# B&R Automation Studio project ciclicheskoe11
Automation Studio 4.5.2.102; technology packages: Acp10Arnc0 1.0.0

## Configuration Config1

CPU 4PP065.0571-P74, AutomationRuntime D4.52, Build 4.1.2, Vc V4.52.0

### Task classes (Cpu.sw)
```
Cyclic#1:
  RobotContr <- RobotControl.prg
DataObjects: Acp10sys
Binaries: TCData, vcfile, vcfntttf, vcpfmtcx, arial, vcmgr, vccovl, vcdsint, vcpdpp30, vcshared, vcpfpp30, vcpdsw, vcalarm, vccbtn, vcptelo, vcgclass, vcdsloc, arialbd, vcrt, Visu02, vctcal, Visu01, Visu03, vcbclass, udbdef, vcctext, vccbmp, vcchspot, vccnum, ashwac, arconfig, User, sysconf, iomap, asfw, ashwd, Role, acp10cfg, Acp10map
Libraries: Acp10sdc, URTK_lib, Acp10man, Acp10par, NcGlobal, asstring, powerlnk, astime, fileio, runtime, dataobj, vcresman, Library
```

### Hardware
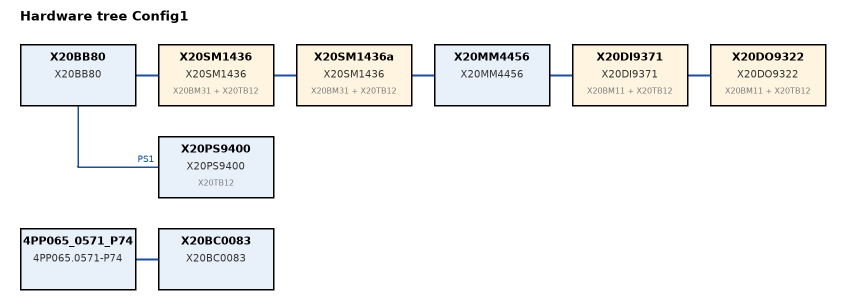
```
4PP065_0571_P74 : 4PP065.0571-P74 v1.1.2.0
  Connector IF4:
    EplInterfaceRedundant = 0
    EplEthInterfaceRedundant = 0
  Connector IF5:
    ActivateDevice = 1
    Mode = Manual
    InternetAddress = 10.0.1.10
    SubnetMask = 255.255.255.0
  ConfigurationID = labBR
  TimerDeviceType = EPLX2X
  TimerDevice = 4PP065_0571_P74.IF4
  TaskClassIdleTime = 2000
  Cyclic1Tolerance = 0
  Cyclic1Output = 1
X20BB80 : X20BB80 v1.0.2.0
X20BC0083 : X20BC0083 v2.7.0.0  [PLK1 -> 4PP065_0571_P74.IF4 (NodeNumber=2) [Cable Type=PowerlinkCable, Length=10, Version=1.0.0.2]; SL -> X20BB80.SL1]
X20BM11 : X20BM11 v1.0.0.1  [X2X1 -> X20MM4456.X2X2]
X20BM11a : X20BM11 v1.0.0.1  [X2X1 -> X20BM11.X2X2]
X20BM31 : X20BM31 v1.0.0.1  [X2X1 -> X20BB80.IF1]
X20BM31a : X20BM31 v1.0.0.1  [X2X1 -> X20BM31.X2X2]
X20DI9371 : X20DI9371 v1.0.2.0  [SS1 -> X20TB12c.SS; SL -> X20BM11.SL1]
X20DO9322 : X20DO9322 v1.0.3.0  [SS1 -> X20TB12d.SS; SL -> X20BM11a.SL1]
X20MM4456 : X20MM4456 v1.1.5.0  [X2X1 -> X20BM31a.X2X2]
X20PS9400 : X20PS9400 v1.0.2.4  [SS1 -> X20TB12.SS; PS -> X20BB80.PS1]
X20SM1436 : X20SM1436 v1.4.2.1  [SS1 -> X20TB12a.SS; SL -> X20BM31.SL1]
X20SM1436a : X20SM1436 v1.4.2.1  [SS1 -> X20TB12b.SS; SL -> X20BM31a.SL1]
X20TB12 : X20TB12 v1.0.0.0
X20TB12a : X20TB12 v1.0.0.0
X20TB12b : X20TB12 v1.0.0.0
X20TB12c : X20TB12 v1.0.0.0
X20TB12d : X20TB12 v1.0.0.0
```

### IoMap.iom - 4PP065_0571_P74/IoMap.iom
```iecst
VAR_CONFIG
	::RobotContr:URTK_Ctrl.AxisX.hardware.PeriodDurationPWM AT %QW."X20MM4456".PeriodDurationPWM;
	::RobotContr:URTK_Ctrl.AxisX.hardware.ShowMeanCurrent AT %QX."X20MM4456".ShowMeanCurrent01;
	::RobotContr:URTK_Ctrl.AxisX.hardware.Counter AT %IW."X20MM4456".Counter01;
	::RobotContr:URTK_Ctrl.AxisX.hardware.CounterLatch AT %IW."X20MM4456".CounterLatch01;
	::RobotContr:URTK_Ctrl.AxisX.hardware.PulseWidthCurrentPWM AT %QW."X20MM4456".PulseWidthCurrentPWM01;
	::RobotContr:URTK_Ctrl.Ustator AT %QW."X20MM4456".PulseWidthCurrentPWM04;
	::RobotContr:URTK_Ctrl.AxisX.hardware.StatusInputP AT %IX."X20MM4456".StatusInput03;
	::RobotContr:URTK_Ctrl.AxisX.hardware.StatusInputN AT %IX."X20MM4456".StatusInput04;
	::RobotContr:URTK_Ctrl.AxisY.hardware.StatusInputP AT %IX."X20MM4456".StatusInput07;
	::RobotContr:URTK_Ctrl.AxisY.hardware.StatusInputN AT %IX."X20MM4456".StatusInput08;
	::RobotContr:URTK_Ctrl.AxisY.hardware.Counter AT %IW."X20MM4456".Counter02;
	::RobotContr:URTK_Ctrl.AxisY.hardware.CounterLatch AT %IW."X20MM4456".CounterLatch02;
	::RobotContr:URTK_Ctrl.AxisY.hardware.ShowMeanCurrent AT %QX."X20MM4456".ShowMeanCurrent02;
	::RobotContr:URTK_Ctrl.AxisY.hardware.PulseWidthCurrentPWM AT %QW."X20MM4456".PulseWidthCurrentPWM02;
	::RobotContr:URTK_Ctrl.AxisZ.hardware.StatusInputP AT %IX."X20MM4456".StatusInput11;
	::RobotContr:URTK_Ctrl.AxisZ.hardware.StatusInputN AT %IX."X20MM4456".StatusInput12;
	::RobotContr:URTK_Ctrl.AxisZ.hardware.Counter AT %IW."X20MM4456".Counter03;
	::RobotContr:URTK_Ctrl.AxisZ.hardware.CounterLatch AT %IW."X20MM4456".CounterLatch03;
	::RobotContr:URTK_Ctrl.AxisZ.hardware.ShowMeanCurrent AT %QX."X20MM4456".ShowMeanCurrent03;
	::RobotContr:URTK_Ctrl.AxisZ.hardware.PulseWidthCurrentPWM AT %QW."X20MM4456".PulseWidthCurrentPWM03;
	::RobotContr:URTK_Ctrl.FBHomingX.ResetCounter AT %QX."X20MM4456".ResetCounter01;
	::RobotContr:URTK_Ctrl.FBHomingY.ResetCounter AT %QX."X20MM4456".ResetCounter02;
	::RobotContr:URTK_Ctrl.FBHomingZ.ResetCounter AT %QX."X20MM4456".ResetCounter03;
	::RobotContr:URTK_Ctrl.Hardware.UnderVoltageError AT %IX."X20MM4456".UnderVoltageError;
	::RobotContr:URTK_Ctrl.Hardware.VoltageWarning AT %IX."X20MM4456".VoltageWarning;
	::RobotContr:URTK_Ctrl.Hardware.OverVoltageError AT %IX."X20MM4456".OverVoltageError;
	::RobotContr:URTK_Ctrl.Hardware.OverTemperatureError AT %IX."X20MM4456".OvertemperatureError;
	::RobotContr:URTK_Ctrl.Hardware.PWMError01 AT %IX."X20MM4456".PWMError01;
	::RobotContr:URTK_Ctrl.Hardware.CurrentError01 AT %IX."X20MM4456".CurrentError01;
	::RobotContr:URTK_Ctrl.Hardware.OverCurrentError01 AT %IX."X20MM4456".OverCurrentError01;
	::RobotContr:URTK_Ctrl.Hardware.CurrentError02 AT %IX."X20MM4456".CurrentError02;
	::RobotContr:URTK_Ctrl.Hardware.CurrentError03 AT %IX."X20MM4456".CurrentError03;
	::RobotContr:URTK_Ctrl.Hardware.OverCurrentError02 AT %IX."X20MM4456".OverCurrentError02;
	::RobotContr:URTK_Ctrl.Hardware.PWMError02 AT %IX."X20MM4456".PWMError02;
	::RobotContr:URTK_Ctrl.Hardware.PWMError03 AT %IX."X20MM4456".PWMError03;
	::RobotContr:URTK_Ctrl.Control.Grip AT %QX."X20DO9322".DigitalOutput01;
	::RobotContr:led1 AT %QX."X20DO9322".DigitalOutput02;
	::RobotContr:led2 AT %QX."X20DO9322".DigitalOutput03;
	::RobotContr:led3 AT %QX."X20DO9322".DigitalOutput04;
	::RobotContr:led4 AT %QX."X20DO9322".DigitalOutput05;
	::RobotContr:BtnS AT %IX."X20DI9371".DigitalInput01;
	::RobotContr:URTK_Ctrl.Hardware.OverCurrentError03 AT %IX."X20MM4456".OverCurrentError03;
END_VAR
```

## Logical view

Binary libraries used (declarations not repeated): operator, runtime, astime, AsIecCon, Acp10sdc, Acp10man, Acp10par, NcGlobal, asstring

### Package Logical/Libraries - Global libraries

### Library Logical/Libraries/Library (ANSIC)

#### Library.fun
```iecst
FUNCTION_BLOCK FB_Motor (*TODO: Add your comment here*) (*$GROUP=User,$CAT=User,$GROUPICON=User.png,$CATICON=User.png*)
	VAR_INPUT
		in : REAL;
	END_VAR
	VAR_OUTPUT
		out_w : REAL;
		out_phi : REAL;
	END_VAR
	VAR
		k_e : REAL;
		T_m : REAL;
		dt : REAL;
		integrator : FB_Integrator;
		integrator_phi : FB_Integrator;
	END_VAR
END_FUNCTION_BLOCK

FUNCTION_BLOCK FB_Integrator (*TODO: Add your comment here*) (*$GROUP=User,$CAT=User,$GROUPICON=User.png,$CATICON=User.png*)
	VAR_INPUT
		in : REAL;
		dt : REAL;
	END_VAR
	VAR_OUTPUT
		out : REAL;
	END_VAR
	VAR
		state : REAL := 0.0;
	END_VAR
END_FUNCTION_BLOCK

FUNCTION_BLOCK FB_Controller (* *) (*$GROUP=User,$CAT=User,$GROUPICON=User.png,$CATICON=User.png*)
	VAR_INPUT
		in : REAL;
		k_i : REAL;
		k_d : REAL;
		k_p : REAL;
		dt : REAL;
	END_VAR
	VAR_OUTPUT
		out : REAL;
	END_VAR
	VAR
		max_abs_value : REAL := 32767;
		prev_in : REAL;
	END_VAR
END_FUNCTION_BLOCK

FUNCTION_BLOCK FB_Endswitch (*TODO: Add your comment here*) (*$GROUP=User,$CAT=User,$GROUPICON=User.png,$CATICON=User.png*)
	VAR_INPUT
		in : REAL;
		neg_value : REAL;
		pos_value : REAL;
	END_VAR
	VAR_OUTPUT
		neg_reached : BOOL;
		pos_reached : BOOL;
	END_VAR
END_FUNCTION_BLOCK

FUNCTION_BLOCK FB_Axis (*TODO: Add your comment here*) (*$GROUP=User,$CAT=User,$GROUPICON=User.png,$CATICON=User.png*)
	VAR_INPUT
		reset_error : BOOL;
		endswitch_a_reached : BOOL;
		endswitch_b_reached : BOOL;
		pwm_percentage : SINT;
	END_VAR
	VAR_OUTPUT
		reset_counter : BOOL;
		pwm_value : INT;
	END_VAR
	VAR_OUTPUT RETAIN
		counter : INT;
	END_VAR
	VAR_OUTPUT
		speed : REAL;
	END_VAR
	VAR
		last_counter : INT;
	END_VAR
END_FUNCTION_BLOCK

{REDUND_ERROR} FUNCTION_BLOCK FB_PD (*TODO: Add your comment here*) (*$GROUP=User,$CAT=User,$GROUPICON=User.png,$CATICON=User.png*)
	VAR_INPUT
		in : {REDUND_UNREPLICABLE} REAL;
		k_d : REAL;
		k_p : REAL;
		dt : REAL;
	END_VAR
	VAR_OUTPUT
		out : REAL;
	END_VAR
	VAR
		max_abs_value : REAL := 32767;
		prev_in : REAL;
	END_VAR
END_FUNCTION_BLOCK
```

#### FB_Controller.c
```c
#include <bur/plctypes.h>
#ifdef __cplusplus
	extern "C"
	{
#endif
	#include "Library.h"
#ifdef __cplusplus
	};
#endif

void FB_Controller(struct FB_Controller* inst)
{
	inst->out = inst->k_p*inst->in + inst->k_d*(inst->in-inst->prev_in)*inst->dt + inst->k_i*(inst->dt * inst->in + inst->prev_in)*inst->dt;
	inst->out = inst->out > inst->max_abs_value ? inst->max_abs_value : inst->out;
	inst->out = inst->out < -inst->max_abs_value ? -inst->max_abs_value : inst->out;
	inst->prev_in = inst->in;
}
```

#### FB_Endswitch.c
```c
#include <bur/plctypes.h>
#ifdef __cplusplus
	extern "C"
	{
#endif
	#include "Library.h"
#ifdef __cplusplus
	};
#endif
/* TODO: Add your comment here */
void FB_Endswitch(struct FB_Endswitch* inst)
{

}
```

#### FB_PD.c
```c
#include <bur/plctypes.h>
#ifdef __cplusplus
	extern "C"
	{
#endif
	#include "Library.h"
#ifdef __cplusplus
	};
#endif
/* TODO: Add your comment here */
void FB_PD(struct FB_PD* inst)
{
	inst->out = inst->k_p*inst->in + inst->k_d*(inst->in-inst->prev_in)*inst->dt;
	//inst->out = inst->k_p*inst->in + inst->k_d*(inst->dt * inst->in + inst->prev_in)*inst->dt;
	inst->out = inst->out > inst->max_abs_value ? inst->max_abs_value : inst->out;
	inst->out = inst->out < -inst->max_abs_value ? -inst->max_abs_value : inst->out;
	inst->prev_in = inst->in;
}
```

### Library Logical/Libraries/URTK_lib (ANSIC)

#### Types.typ - Exported data types
```iecst
TYPE
	TURTKAxisMonitor : 	STRUCT
		Position : REAL;
		LimitN : BOOL;
		LimitP : BOOL;
		Iact : REAL; (*Измеряемый ток в амперах*)
		Uact : REAL; (*Фактически формируемое напряжение*)
	END_STRUCT;
	TURTKAxicCtrl : 	STRUCT
		U : REAL; (*напряжение в вольтах*)
		ILim : REAL; (*ограничение тока в Амперах*)
		ClearError : BOOL;
	END_STRUCT;
	TURTKAxisError : 	STRUCT
		OverCurrent : BOOL;
	END_STRUCT;
	TURTKAxisHardware : 	STRUCT
		PeriodDurationPWM : UINT := 20;
		StatusInputP : BOOL;
		StatusInputN : BOOL;
		PulseWidthCurrentPWM : INT;
		ShowMeanCurrent : BOOL;
		Counter : INT;
		CounterLatch : INT;
	END_STRUCT;
	TURTKHomingState :
		(
		ST_IDLE,
		ST_MOVE_FAST,
		ST_MOVE_SLOW
		);
	TURTKMovePos :
		(
		ST_IDLE_POS,
		ST_MOVE_POS
		);
	TURTKHardware : 	STRUCT
		PWMDuration : UINT;
		PWMX : INT;
		Error : BOOL;
		Grip : BOOL;
		UnderVoltageError : BOOL;
		VoltageWarning : BOOL;
		OverVoltageError : BOOL;
		OverTemperatureError : BOOL;
		PWMError01 : BOOL;
		CurrentError01 : BOOL;
		OverCurrentError01 : BOOL;
		PWMError02 : BOOL;
		CurrentError02 : BOOL;
		OverCurrentError02 : BOOL;
		PWMError03 : BOOL;
		CurrentError03 : BOOL;
		OverCurrentError03 : BOOL;
	END_STRUCT;
	ERROR :
		(
		ERR_URTK_NO_ERROR := 0,
		ERR_URTK_UNDERVOLTAGE := 1,
		ERR_URTK_VOLTAGEWARNING := 3,
		ERR_URTK_OVERVOLTAGE := 4,
		ERR_URTK_OVERTEMPERATURE := 5,
		ERR_URTK_PWM01 := 6,
		ERR_URTK_CURRENT01 := 7,
		ERR_URTK_OVERCURRENT01 := 8,
		ERR_URTK_PWM02 := 9,
		ERR_URTK_CURRENT02 := 10,
		ERR_URTK_OVERCURRENT02 := 11,
		ERR_URTK_PWM03 := 12,
		ERR_URTK_CURRENT03 := 13,
		ERR_URTK_OVERCURRENT03 := 14
		);
	TURTKMonitor : 	STRUCT
		PositionX : REAL;
		PositionY : REAL;
		PositionZ : REAL;
		LimitX_N : BOOL;
		LimitX_P : BOOL;
		LimitY_N : BOOL;
		LimitY_P : BOOL;
		LimitZ_N : BOOL;
		LimitZ_P : BOOL;
		Grip : BOOL;
		HomingX : FB_URTKAxisHome;
		HomingY : FB_URTKAxisHome;
		HomingZ : FB_URTKAxisHome;
		HomingOK : BOOL;
		InPosition : BOOL;
	END_STRUCT;
	TURTKError : 	STRUCT
		Type : ERROR;
		Error : BOOL;
		CLearError : BOOL;
		ConfigIun : BOOL;
		prevCLearError : BOOL;
	END_STRUCT;
	TURTKControl : 	STRUCT
		ManualCtrl : BOOL;
		StartHoming : BOOL;
		MovPos : BOOL;
		X : REAL;
		Y : REAL;
		Z : REAL;
		ManBtnXPos : BOOL;
		ManBtnXNeg : BOOL;
		ManBtnYPos : BOOL;
		ManBtnYNeg : BOOL;
		ManBtnZPos : BOOL;
		ManBtnZNeg : BOOL;
		Grip : BOOL;
	END_STRUCT;
	URTKCtrl :
		(
		ST_URTK_IDLE,
		ST_URTK_MANUAL,
		ST_URTK_ERROR,
		ST_URTK_HOMING,
		ST_URTK_MOVE_POS,
		ST_POS1,
		ST_POS2,
		ST_POS3
		);
END_TYPE
```

#### URTK_lib.fun - Exported functions and function blocks
```iecst
FUNCTION_BLOCK FBURTKAxis (*функциональный блок управления одной степенью *) (*$GROUP=User,$CAT=User,$GROUPICON=User.png,$CATICON=User.png*)
	VAR_INPUT
		control : TURTKAxicCtrl;
		monitor : TURTKAxisMonitor;
		error : TURTKAxisError;
		hardware : TURTKAxisHardware;
	END_VAR
END_FUNCTION_BLOCK

FUNCTION_BLOCK FB_URTKAxisHome (*TODO: Add your comment here*) (*$GROUP=User,$CAT=User,$GROUPICON=User.png,$CATICON=User.png*)
	VAR_INPUT
		U_fast : REAL;
		U_low : REAL;
		pos_direction : BOOL;
		LimitP : BOOL;
		LimitN : BOOL;
		enable : BOOL;
	END_VAR
	VAR_OUTPUT
		U : REAL;
		done : BOOL;
		ResetCounter : BOOL;
		State : TURTKHomingState;
	END_VAR
	VAR
		p_dir : BOOL;
	END_VAR
END_FUNCTION_BLOCK

FUNCTION_BLOCK FBURTKAxisMovePos (*TODO: Add your comment here*) (*$GROUP=User,$CAT=User,$GROUPICON=User.png,$CATICON=User.png*)
	VAR_INPUT
		set_position : REAL;
		set_position1 : REAL;
		set_position2 : REAL;
		act_position : REAL;
		homing_done : BOOL;
		K : REAL;
		enable : BOOL;
	END_VAR
	VAR_OUTPUT
		done : BOOL;
		U : REAL;
		State : TURTKMovePos;
		done1 : BOOL;
		done2 : BOOL;
		done3 : BOOL;
	END_VAR
END_FUNCTION_BLOCK

FUNCTION_BLOCK FBURTKCtrl (*TODO: Add your comment here*) (*$GROUP=User,$CAT=User,$GROUPICON=User.png,$CATICON=User.png*)
	VAR_INPUT
		Grip : BOOL;
		Hardware : TURTKHardware;
		Monitor : TURTKMonitor;
		Error : TURTKError;
		Control : TURTKControl;
		enable : BOOL;
		AxisX : FBURTKAxis;
		AxisY : FBURTKAxis;
		AxisZ : FBURTKAxis;
		FBHomingX : FB_URTKAxisHome;
		FBHomingY : FB_URTKAxisHome;
		FBHomingZ : FB_URTKAxisHome;
		FBMovePosX : FBURTKAxisMovePos;
		FBMovePosY : FBURTKAxisMovePos;
		FBMovePosZ : FBURTKAxisMovePos;
		Ustator : INT;
	END_VAR
	VAR_OUTPUT
		State : URTKCtrl;
	END_VAR
END_FUNCTION_BLOCK
```

#### FBURTKAxis.c
```c
#include <bur/plctypes.h>
#ifdef __cplusplus
	extern "C"
	{
#endif
	#include "URTK_lib.h"
#ifdef __cplusplus
	};
#endif
/* функциональный блок управления одной степенью  */
void FBURTKAxis(struct FBURTKAxis* inst)
{
	//Обработка переменных мониторинга
	inst->hardware.PeriodDurationPWM=20;//Устанавливаем период ШИМ 20 мкс
	inst->hardware.ShowMeanCurrent=1;   //Включаем измерение тока
	inst->monitor.Iact=inst->hardware.CounterLatch;
	inst->monitor.Iact=inst->monitor.Iact/32767*10;
	inst->monitor.Position=inst->hardware.Counter;
	inst->monitor.Position=inst->monitor.Position/24*3; // 3 мм/об / 24 метки/об
	inst->monitor.LimitN=inst->hardware.StatusInputN;
	inst->monitor.LimitP=inst->hardware.StatusInputP;

	//Обработка ошибок
	if(((inst->monitor.Iact>0)&&(inst->monitor.Iact>inst->control.ILim))||
	   ((inst->monitor.Iact<0)&&(inst->monitor.Iact<-inst->control.ILim)))
		inst->error.OverCurrent=1;
	if(inst->control.ClearError)
		inst->error.OverCurrent=0;

	//Проверка ограничений
	inst->monitor.Uact=inst->control.U;
	if(inst->error.OverCurrent)
		inst->monitor.Uact = 0;
	if(inst->monitor.LimitN&&(inst->monitor.Uact<=0))
		inst->monitor.Uact = 0;
	if(inst->monitor.LimitP&&(inst->monitor.Uact>=0))
		inst->monitor.Uact = 0;
	if(inst->monitor.Uact>24.0)
		inst->monitor.Uact=24.0;
	if(inst->monitor.Uact<-24.0)
		inst->monitor.Uact=-24.0;

	//Формирование выходного сигнала
	inst->hardware.PulseWidthCurrentPWM=inst->monitor.Uact/24.0*32767.0;

}
```

#### FB_URTKAxisHome.c
```c
#include <bur/plctypes.h>
#ifdef __cplusplus
	extern "C"
	{
#endif
	#include "URTK_lib.h"
#ifdef __cplusplus
	};
#endif
/* функциональный блок */
void FB_URTKAxisHome(struct FB_URTKAxisHome* inst)
{
	switch (inst->State){
		case ST_IDLE:
			inst->U=0;
			inst->ResetCounter=0;
			if(inst->enable){
				inst->p_dir=inst->pos_direction;
				inst->State=ST_MOVE_FAST;
				inst->done=0;
			}

		case ST_MOVE_FAST:
			if(!inst->enable){
				inst->U=0;
				inst->ResetCounter=0;
				inst->State=ST_IDLE;
			}

			if(inst->p_dir){
			inst->ResetCounter = 0;
			inst->U=inst->U_fast;
			}
			else{
			inst->ResetCounter = 0;
			inst->U=-inst->U_fast;
			}

			if(inst->LimitN||inst->LimitP){
			inst->U=0;
			inst->ResetCounter=0;
			inst->State=ST_MOVE_SLOW;
			}
			break;

		case ST_MOVE_SLOW:
			if(!inst->enable){
				inst->U=0;
				inst->ResetCounter=0;
				inst->State=ST_IDLE;
			}

	/*		if(inst->ResetCounter == (!inst->LimitP))
				inst->U=-inst->U_low;

			if(inst->ResetCounter == (!inst->LimitN))
				inst->U=8;
*/
			if(inst->p_dir=1){
			inst->ResetCounter = (!inst->LimitP);
			inst->U = 6;

			}

			if(inst->p_dir=0){

				inst->ResetCounter = (!inst->LimitN);
				inst->U = inst->U_low;
			}
		/*	else{

				inst->ResetCounter = (!inst->LimitN);
				inst->U = inst->U_low;

			}*/

			if(!(inst->LimitN||inst->LimitP)){
			inst->State=ST_IDLE;
			inst->enable=0;
			inst->done=1;
			}
			break;

	}
}
```

#### FBURTKAxisMovePos.c
```c
#include <bur/plctypes.h>
#ifdef __cplusplus
	extern "C"
	{
#endif
	#include "URTK_lib.h"
#ifdef __cplusplus
	};
#endif
/* TODO: Add your comment here */
void FBURTKAxisMovePos(struct FBURTKAxisMovePos* inst)
{
	inst->done=(inst->set_position==inst->act_position);
	switch (inst->State){
		case ST_IDLE_POS:
			inst->U=0;
		//	inst->act_position=0; //где мы есть
			if(inst->enable){
				inst->State=ST_MOVE_POS;
				if(!inst->homing_done){
					inst->State=ST_IDLE_POS;
					inst->enable=0;
				}
			}
			break;
		case ST_MOVE_POS:
			if(!inst->enable){
				inst->U=0;
				inst->State=ST_IDLE_POS;
			}
			inst->U=inst->K*((inst->set_position)-(inst->act_position));
			if(inst->U > 14)
			{
				inst->U = 14;
			}
			if(inst->done){
				inst->State=ST_IDLE_POS;
				inst->enable=0;
			}
			break;
	}
}
```

#### FBURTKCtrl.c
```c
#include <bur/plctypes.h>
#ifdef __cplusplus
	extern "C"
	{
#endif
	#include "URTK_lib.h"
#ifdef __cplusplus
	};
#endif
/* TODO: Add your comment here */
void FBURTKCtrl(struct FBURTKCtrl* inst)
{
	FBURTKAxis(&inst->AxisX);
	FBURTKAxis(&inst->AxisY);
	FBURTKAxis(&inst->AxisZ);
//	FBERROR(&inst->Error1);

	if(inst->Hardware.UnderVoltageError){
		inst->Error.Error=1;
		inst->Error.Type=ERR_URTK_UNDERVOLTAGE;
		inst->Ustator=0;
	}
	if(inst->Hardware.VoltageWarning){
		inst->Error.Error=1;
		inst->Error.Type=ERR_URTK_VOLTAGEWARNING;
		inst->Ustator=0;
	}
	if(inst->Hardware.OverVoltageError){
		inst->Error.Error=1;
		inst->Error.Type=ERR_URTK_OVERVOLTAGE;
		inst->Ustator=0;
	}
	if(inst->Hardware.OverTemperatureError){
		inst->Error.Error=1;
		inst->Error.Type=ERR_URTK_OVERTEMPERATURE;
		inst->Ustator=0;
	}
	if(inst->Hardware.PWMError01){
		inst->Error.Error=1;
		inst->Error.Type=ERR_URTK_PWM01;
		inst->Ustator=0;
	}
	if(inst->Hardware.CurrentError01){
		inst->Error.Error=1;
		inst->Error.Type=ERR_URTK_CURRENT01;
		inst->Ustator=0;
	}
	if(inst->Hardware.OverCurrentError01){
		inst->Error.Error=1;
		inst->Error.Type=ERR_URTK_OVERCURRENT01;
		inst->Ustator=0;
	}
	if(inst->Hardware.PWMError02){
		inst->Error.Error=1;
		inst->Error.Type=ERR_URTK_PWM02;
		inst->Ustator=0;
	}
	if(inst->Hardware.CurrentError02){
		inst->Error.Error=1;
		inst->Error.Type=ERR_URTK_CURRENT02;
		inst->Ustator=0;
	}
	if(inst->Hardware.OverCurrentError02){
		inst->Error.Error=1;
		inst->Error.Type=ERR_URTK_OVERCURRENT02;
		inst->Ustator=0;
	}
	if(inst->Hardware.PWMError03){
		inst->Error.Error=1;
		inst->Error.Type=ERR_URTK_PWM03;
		inst->Ustator=0;
	}
	if(inst->Hardware.CurrentError03){
		inst->Error.Error=1;
		inst->Error.Type=ERR_URTK_CURRENT03;
		inst->Ustator=0;
	}
	if(inst->Hardware.OverCurrentError03){
		inst->Error.Error=1;
		inst->Error.Type=ERR_URTK_OVERCURRENT03;
		inst->Ustator=0;
	}
	if(!inst->Error.Error){//if(!inst->Hardware.Error)
		inst->Error.Error=0;// не было
		inst->Error.Type=ERR_URTK_NO_ERROR;
		inst->Error.CLearError=0;
	}

	if(inst->Error.CLearError&(!inst->Error.prevCLearError)){
		switch (inst->Error.Type){
			case ERR_URTK_UNDERVOLTAGE:
				inst->Error.Error=0;
				inst->Error.Type=ERR_URTK_NO_ERROR;
				break;

			case ERR_URTK_VOLTAGEWARNING:
				inst->Error.Error=0;
				inst->Error.Type=ERR_URTK_NO_ERROR;
				break;

			case ERR_URTK_OVERVOLTAGE:
				inst->Error.Error=0;
				inst->Error.Type=ERR_URTK_NO_ERROR;
				break;

			case ERR_URTK_OVERTEMPERATURE:
				inst->Error.Error=0;
				inst->Error.Type=ERR_URTK_NO_ERROR;
				break;

			case ERR_URTK_PWM01:
				inst->Error.Error=0;
				inst->Error.Type=ERR_URTK_NO_ERROR;
				break;

			case ERR_URTK_CURRENT01:
				inst->Error.Error=0;
				inst->Error.Type=ERR_URTK_NO_ERROR;
				break;

			case ERR_URTK_OVERCURRENT01:
				inst->Error.Error=0;
				inst->Error.Type=ERR_URTK_NO_ERROR;
				break;

			case ERR_URTK_PWM02:
				inst->Error.Error=0;
				inst->Error.Type=ERR_URTK_NO_ERROR;
				break;

			case ERR_URTK_CURRENT02:
				inst->Error.Error=0;
				inst->Error.Type=ERR_URTK_NO_ERROR;
				break;

			case ERR_URTK_OVERCURRENT02:
				inst->Error.Error=0;
				inst->Error.Type=ERR_URTK_NO_ERROR;
				break;

			case ERR_URTK_PWM03:
				inst->Error.Error=0;
				inst->Error.Type=ERR_URTK_NO_ERROR;
				break;

			case ERR_URTK_CURRENT03:
				inst->Error.Error=0;
				inst->Error.Type=ERR_URTK_NO_ERROR;
				break;

			case ERR_URTK_OVERCURRENT03:
				inst->Error.Error=0;
				inst->Error.Type=ERR_URTK_NO_ERROR;
				break;
		}

	}

	switch (inst->State){
		case ST_URTK_IDLE:

			//	inst->AxisX.hardware.PeriodDurationPWM = 32767;

			inst->enable=1;

			inst->Ustator=0;

			inst->AxisX.control.U=0;
			inst->AxisY.control.U=0;
			inst->AxisZ.control.U=0;

			//		inst->FBMovePosX.set_position=10;  //задание точек
			//		inst->FBMovePosY.set_position=15;
			//		inst->FBMovePosZ.set_position=30;
			//		inst->FBMovePosX.set_position1=70;
			//		inst->FBMovePosY.set_position1=60;
			//		inst->FBMovePosZ.set_position1=60;
			//		inst->FBMovePosX.set_position2=30;
			//		inst->FBMovePosY.set_position2=40;
			//		inst->FBMovePosZ.set_position2=25;

			//	inst->FBMovePosX.set_position=inst->Control.X;
			//	inst->FBMovePosY.set_position=inst->Control.Y;
			//	inst->FBMovePosZ.set_position=inst->Control.Z;

			if(inst->Control.MovPos){
				inst->FBMovePosX.set_position=10;  //задание точек
				inst->FBMovePosY.set_position=15;
				inst->FBMovePosZ.set_position=30;
				inst->FBMovePosX.act_position=0;
				inst->FBMovePosY.act_position=0;
				inst->FBMovePosZ.act_position=0;
				inst->FBMovePosX.enable=inst->enable;
				inst->FBMovePosY.enable=inst->enable;
				inst->FBMovePosZ.enable=inst->enable;
				inst->FBMovePosX.homing_done=1;
				inst->FBMovePosY.homing_done=1;
				inst->FBMovePosZ.homing_done=1;
				//	inst->Ustator=32767;
				inst->State=ST_URTK_MOVE_POS;
				break;
			/*	if(inst->Monitor.HomingOK){
					inst->FBMovePosX.set_position=10;  //задание точек
					inst->FBMovePosY.set_position=15;
					inst->FBMovePosZ.set_position=30;
					inst->FBMovePosX.act_position=0;
					inst->FBMovePosY.act_position=0;
					inst->FBMovePosZ.act_position=0;
					inst->FBMovePosX.enable=inst->enable;
					inst->FBMovePosY.enable=inst->enable;
					inst->FBMovePosZ.enable=inst->enable;
					inst->FBMovePosX.homing_done=1;
					inst->FBMovePosY.homing_done=1;
					inst->FBMovePosZ.homing_done=1;
				//	inst->Ustator=32767;
					inst->State=ST_URTK_MOVE_POS;
					break;
				}*/
			}
			if(inst->Control.StartHoming){
				inst->FBHomingX.enable=inst->enable;
				inst->FBHomingY.enable=inst->enable;
				inst->FBHomingZ.enable=inst->enable;
				//		inst->Ustator=32767;
				inst->State=ST_URTK_HOMING;
				break;
			}
			if(inst->Control.ManualCtrl){
				//		inst->Ustator=32767;
				inst->State=ST_URTK_MANUAL;
				break;
			}
			break;

		case ST_URTK_MANUAL:

			inst->AxisX.control.U=0;
			inst->AxisY.control.U=0;
			inst->AxisZ.control.U=0;

			if(inst->Control.ManBtnXPos){
				inst->AxisX.control.U=18.0;		//переменная управления движком
			}
			if(inst->Control.ManBtnXNeg){
				inst->AxisX.control.U=-18.0;
			}

			if(inst->Control.ManBtnYPos){
				inst->AxisY.control.U=18.0;
			}
			if(inst->Control.ManBtnYNeg){
				inst->AxisY.control.U=-18.0;
			}

			if(inst->Control.ManBtnZPos){
				inst->AxisZ.control.U=18.0;
			}
			if(inst->Control.ManBtnZNeg){
				inst->AxisZ.control.U=-18.0;
			}

			if(!inst->Control.ManualCtrl){
				inst->Ustator=0;
				inst->State=ST_URTK_IDLE;
				break;
			}
			break;

		case ST_URTK_HOMING:
			inst->FBHomingX.LimitN = inst->AxisX.hardware.StatusInputN;
			inst->FBHomingX.LimitP = inst->AxisX.hardware.StatusInputP;
			if(!inst->FBHomingX.done){
				inst->AxisX.control.U = inst->FBHomingX.U;
			}

			inst->FBHomingY.LimitN = inst->AxisY.hardware.StatusInputN;
			inst->FBHomingY.LimitP = inst->AxisY.hardware.StatusInputP;
			if(!inst->FBHomingY.done){
				inst->AxisY.control.U = inst->FBHomingY.U;
			}

			inst->FBHomingZ.LimitN = inst->AxisZ.hardware.StatusInputN;
			inst->FBHomingZ.LimitP = inst->AxisZ.hardware.StatusInputP;
			if(!inst->FBHomingZ.done){
				inst->AxisZ.control.U = inst->FBHomingZ.U;
			}

			if(inst->FBHomingX.done){
				inst->AxisX.control.U = 0;
				inst->FBHomingX.enable=0;
				//		inst->FBHomingX.done=inst->Monitor.HomingX.done;//
			}
			if(inst->FBHomingY.done){
				inst->AxisY.control.U = 0;
				inst->FBHomingY.enable=0;
				//		inst->FBHomingY.done=inst->Monitor.HomingY.done;//
			}
			if(inst->FBHomingZ.done){
				inst->AxisZ.control.U = 0;
				inst->FBHomingZ.enable=0;
				//	inst->FBHomingZ.done=inst->Monitor.HomingZ.done;//

			}

			if(inst->FBHomingX.done){
				if(inst->FBHomingY.done){
					if(inst->FBHomingZ.done){
						inst->Monitor.HomingOK=1;
						inst->Ustator=0;
						inst->State=ST_URTK_IDLE;
						inst->Control.StartHoming=!inst->Control.StartHoming;
						inst->FBHomingX.done=0;
						inst->FBHomingY.done=0;
						inst->FBHomingZ.done=0;
					}
				}
			}

			if(!inst->Control.StartHoming){
				inst->Ustator=0;
				inst->State=ST_URTK_IDLE;
				break;
			}

			break;

		case ST_URTK_MOVE_POS:

			if(!inst->FBMovePosX.enable){
				if(!inst->FBMovePosY.enable){
					if(!inst->FBMovePosZ.enable){
						inst->FBMovePosX.enable=inst->enable;
						inst->FBMovePosY.enable=inst->enable;
						inst->FBMovePosZ.enable=inst->enable;
						inst->FBMovePosX.act_position=10;
						inst->FBMovePosY.act_position=15;
						inst->FBMovePosZ.act_position=30;
						inst->State=ST_POS1;
						//					inst->FBMovePosX.U=0;
						//					inst->FBMovePosY.U=0;
						//					inst->FBMovePosZ.U=0;
						inst->FBMovePosX.set_position=70;
						inst->FBMovePosY.set_position=60;
						inst->FBMovePosZ.set_position=60;
						//					inst->FBMovePosX.homing_done=0;
						//					inst->FBMovePosY.homing_done=0;
						//					inst->FBMovePosZ.homing_done=0;
						//					inst->Ustator=0;
						//					inst->Control.MovPos=!inst->Control.MovPos;

					}
				}
			}
			if(!inst->Control.MovPos){
				inst->State=ST_URTK_IDLE;
				inst->FBMovePosX.homing_done=0;
				inst->FBMovePosY.homing_done=0;
				inst->FBMovePosZ.homing_done=0;
				inst->Ustator=0;

				break;
			}

			inst->FBMovePosX.act_position=inst->AxisX.monitor.Position;
			if(inst->FBMovePosX.set_position==10){
				inst->AxisX.control.U = inst->FBMovePosX.U;
			}

			inst->FBMovePosY.act_position=inst->AxisY.monitor.Position;
			if(inst->FBMovePosY.set_position==15){
				inst->AxisY.control.U = inst->FBMovePosY.U;
			}

			inst->FBMovePosZ.act_position=inst->AxisZ.monitor.Position;
			if(inst->FBMovePosZ.set_position==30){
				inst->AxisZ.control.U = -inst->FBMovePosZ.U;
			}

			break;

		case ST_POS1:
			if(!inst->FBMovePosX.enable){
				if(!inst->FBMovePosY.enable){
					if(!inst->FBMovePosZ.enable){
						inst->FBMovePosX.enable=inst->enable;
						inst->FBMovePosY.enable=inst->enable;
						inst->FBMovePosZ.enable=inst->enable;
						inst->FBMovePosX.set_position=30;
						inst->FBMovePosY.set_position=40;
						inst->FBMovePosZ.set_position=40;
						inst->FBMovePosX.act_position=70;
						inst->FBMovePosY.act_position=60;
						inst->FBMovePosZ.act_position=60;
						inst->State=ST_POS2;
						//					inst->FBMovePosX.U=0;
						//					inst->FBMovePosY.U=0;
						//					inst->FBMovePosZ.U=0;

						//					inst->FBMovePosX.homing_done=0;
						//					inst->FBMovePosY.homing_done=0;
						//					inst->FBMovePosZ.homing_done=0;
						//					inst->Ustator=0;
						//					inst->Control.MovPos=!inst->Control.MovPos;

					}
				}
			}
			if(!inst->Control.MovPos){
				inst->State=ST_URTK_IDLE;
				inst->FBMovePosX.homing_done=0;
				inst->FBMovePosY.homing_done=0;
				inst->FBMovePosZ.homing_done=0;
				inst->Ustator=0;

				break;
			}

			inst->FBMovePosX.act_position=inst->AxisX.monitor.Position;
			if(inst->FBMovePosX.set_position==70){
				inst->AxisX.control.U = inst->FBMovePosX.U;
			}

			inst->FBMovePosY.act_position=inst->AxisY.monitor.Position;
			if(inst->FBMovePosY.set_position==60){
				inst->AxisY.control.U = inst->FBMovePosY.U;
			}

			inst->FBMovePosZ.act_position=inst->AxisZ.monitor.Position;
			if(inst->FBMovePosZ.set_position==60){
				inst->AxisZ.control.U = -inst->FBMovePosZ.U;
			}

			break;

		case ST_POS2:

			if(!inst->FBMovePosX.enable){
				if(!inst->FBMovePosY.enable){
					if(!inst->FBMovePosZ.enable){
						inst->FBMovePosX.enable=inst->enable;
						inst->FBMovePosY.enable=inst->enable;
						inst->FBMovePosZ.enable=inst->enable;
						inst->FBMovePosX.set_position=10;  //задание точек
						inst->FBMovePosY.set_position=15;
						inst->FBMovePosZ.set_position=30;
						inst->FBMovePosX.act_position=30;
						inst->FBMovePosY.act_position=40;
						inst->FBMovePosZ.act_position=40;
						inst->State=ST_POS3;
						//				inst->FBMovePosX.U=0;
						//				inst->FBMovePosY.U=0;
						//				inst->FBMovePosZ.U=0;
						//	inst->FBMovePosX.homing_done=0;
						//	inst->FBMovePosY.homing_done=0;
						//	inst->FBMovePosZ.homing_done=0;
						//	inst->Ustator=0;
						//	inst->Control.MovPos=!inst->Control.MovPos;

					}
				}
			}
			if(!inst->Control.MovPos){
				inst->State=ST_URTK_IDLE;
				inst->FBMovePosX.homing_done=0;
				inst->FBMovePosY.homing_done=0;
				inst->FBMovePosZ.homing_done=0;
				inst->Ustator=0;

				break;
			}

			inst->FBMovePosX.act_position=inst->AxisX.monitor.Position;
			if(inst->FBMovePosX.set_position==30){
				inst->AxisX.control.U = -inst->FBMovePosX.U;
			}

			inst->FBMovePosY.act_position=inst->AxisY.monitor.Position;
			if(inst->FBMovePosY.set_position==40){
				inst->AxisY.control.U = -inst->FBMovePosY.U;
			}

			inst->FBMovePosZ.act_position=inst->AxisZ.monitor.Position;
			if(inst->FBMovePosZ.set_position==40){
				inst->AxisZ.control.U = inst->FBMovePosZ.U;
			}

			break;

		case ST_POS3:

			inst->FBMovePosX.enable=1;
			inst->FBMovePosY.enable=1;
			inst->FBMovePosZ.enable=1;

			if(!inst->FBMovePosX.enable){
				if(!inst->FBMovePosY.enable){
					if(!inst->FBMovePosZ.enable){
						inst->FBMovePosX.enable=inst->enable;
						inst->FBMovePosY.enable=inst->enable;
						inst->FBMovePosZ.enable=inst->enable;
						inst->FBMovePosX.set_position=70;  //задание точек
						inst->FBMovePosY.set_position=60;
						inst->FBMovePosZ.set_position=60;
						inst->FBMovePosX.act_position=10;
						inst->FBMovePosY.act_position=15;
						inst->FBMovePosZ.act_position=30;
						inst->State=ST_POS1;
						//				inst->FBMovePosX.U=0;
						//				inst->FBMovePosY.U=0;
						//				inst->FBMovePosZ.U=0;
						//	inst->FBMovePosX.homing_done=0;
						//	inst->FBMovePosY.homing_done=0;
						//	inst->FBMovePosZ.homing_done=0;
						//	inst->Ustator=0;
						//	inst->Control.MovPos=!inst->Control.MovPos;

					}
				}
			}
			if(!inst->Control.MovPos){
				inst->State=ST_URTK_IDLE;
				inst->FBMovePosX.homing_done=0;
				inst->FBMovePosY.homing_done=0;
				inst->FBMovePosZ.homing_done=0;
				inst->Ustator=0;

				break;
			}

			inst->FBMovePosX.act_position=inst->AxisX.monitor.Position;
			if(inst->FBMovePosX.set_position==10){
				inst->AxisX.control.U = -inst->FBMovePosX.U;
			}

			inst->FBMovePosY.act_position=inst->AxisY.monitor.Position;
			if(inst->FBMovePosY.set_position==15){
				inst->AxisY.control.U = -inst->FBMovePosY.U;
			}

			inst->FBMovePosZ.act_position=inst->AxisZ.monitor.Position;
			if(inst->FBMovePosZ.set_position==30){
				inst->AxisZ.control.U = inst->FBMovePosZ.U;
			}

			break;

	}

	FB_URTKAxisHome(&inst->FBHomingX);
	FB_URTKAxisHome(&inst->FBHomingY);
	FB_URTKAxisHome(&inst->FBHomingZ);
	FBURTKAxisMovePos(&inst->FBMovePosX);
	FBURTKAxisMovePos(&inst->FBMovePosY);
	FBURTKAxisMovePos(&inst->FBMovePosZ);
	FBURTKAxis(&inst->AxisX);
	FBURTKAxis(&inst->AxisY);
	FBURTKAxis(&inst->AxisZ);

	inst->Error.prevCLearError=inst->Error.CLearError;

}
```

### Program Logical/RobotControl (ANSIC)

#### Main.c - Init, cyclic, exit code
```c
#include <bur/plctypes.h>

#ifdef _DEFAULT_INCLUDES
	#include <AsDefault.h>
#endif

void _INIT ProgramInit(void)
{
	// Insert code here

	URTK_Ctrl.AxisX.control.ILim=2.5;
	URTK_Ctrl.AxisY.control.ILim=2.5;
	URTK_Ctrl.AxisZ.control.ILim=2.5;
//	URTKAxisHome.State=ST_IDLE;

	URTK_Ctrl.FBHomingX.U_fast=18.0;
	URTK_Ctrl.FBHomingX.U_low=6.0;
	URTK_Ctrl.FBHomingX.pos_direction=0;

//	URTKAxisHomeY.State=ST_IDLE;
	URTK_Ctrl.FBHomingY.U_fast=18.0;
	URTK_Ctrl.FBHomingY.U_low=6.0;
	URTK_Ctrl.FBHomingY.pos_direction=0;

//	URTKAxisHomeZ.State=ST_IDLE;
	URTK_Ctrl.FBHomingZ.U_fast=18.0;
	URTK_Ctrl.FBHomingZ.U_low=6.0;
	URTK_Ctrl.FBHomingZ.pos_direction=0;

	URTK_Ctrl.FBMovePosX.U=0;
	URTK_Ctrl.FBMovePosX.K=18;
	URTK_Ctrl.FBMovePosY.U=0;
	URTK_Ctrl.FBMovePosY.K=18;
	URTK_Ctrl.FBMovePosZ.U=0;
	URTK_Ctrl.FBMovePosZ.K=18;

	URTK_Ctrl.Monitor.HomingOK=0;
	URTK_Ctrl.Ustator=0;

	URTK_Ctrl.FBMovePosX.set_position=0;
	URTK_Ctrl.FBMovePosY.set_position=0;
	URTK_Ctrl.FBMovePosZ.set_position=0;

	pd.k_p = 90;
	pd.k_d = 10;
	pd.dt = 0.01;
	pid.k_p = 37;
	pid.k_i = 80;
	pid.k_d = 2;
	pid.dt = 0.01;

}

void _CYCLIC ProgramCyclic(void)
{

	//	URTKAx.control.U=0;
	//	URTKAy.control.U=0;
	//	URTKAz.control.U=0;

	/*	if(BtnS){
	Ustator=32767;
	}
	if(BtnP){
	URTKAx.control.U=18.0;		//переменная управления движком
	}
	if(BtnN){
	URTKAx.control.U=-18.0;
	}

	if(BtnPY){
	URTKAy.control.U=18.0;
	}
	if(BtnNY){
	URTKAy.control.U=-18.0;
	}

	if(BtnPZ){
	URTKAz.control.U=18.0;
	}
	if(BtnNZ){
	URTKAz.control.U=-18.0;
	}

	URTKAxisHome.LimitN = URTKAx.hardware.StatusInputN; //калибровка начало
	URTKAxisHome.LimitP = URTKAx.hardware.StatusInputP; //проверка на концевой датчик
	FB_URTKAxisHome(&URTKAxisHome); 		//вызов функции калибровки
	if(URTKAxisHome.enable)					//проверка на энейбл сработал или нет
	URTKAx.control.U = URTKAxisHome.U; //запуск мотора через УРТКх

	URTKAxisHomeY.LimitN = URTKAy.hardware.StatusInputN;
	URTKAxisHomeY.LimitP = URTKAy.hardware.StatusInputP;
	FB_URTKAxisHome(&URTKAxisHomeY);
	if(URTKAxisHomeY.enable)
	URTKAy.control.U = URTKAxisHomeY.U;

	URTKAxisHomeZ.LimitN = URTKAz.hardware.StatusInputN;
	URTKAxisHomeZ.LimitP = URTKAz.hardware.StatusInputP;
	FB_URTKAxisHome(&URTKAxisHomeZ);
	if(URTKAxisHomeZ.enable)
	URTKAz.control.U = URTKAxisHomeZ.U; //калибровка конец

	FBURTKAxisMovePos(&URTKAxisMovePos);
	FBURTKAxisMovePos(&URTKAxisMovePosY);
	FBURTKAxisMovePos(&URTKAxisMovePosZ);

	FBURTKAxis(&URTKAx);
	FBURTKAxis(&URTKAy);
	FBURTKAxis(&URTKAz);
	FBURTKAxis(&URTKAt);

	URTKAxisMovePos.homing_done=URTKAxisHome.done;  			//присвоение homing_done заначения done служит для последующего запуска ФБ
	URTKAxisMovePos.act_position=URTKAx.monitor.Position; 		//снятие данных с монитора и запись оных в переменную нынешнего положения
	FBURTKAxisMovePos(&URTKAxisMovePos); 						//вызов функционального блока на переменную
	if(URTKAxisMovePos.enable) 									//проверка на энейбл
	URTKAx.control.U = URTKAxisMovePos.U; 					//запуск двигателя через УРТКх

	URTKAxisMovePosY.homing_done=URTKAxisHomeY.done;
	URTKAxisMovePosY.act_position=URTKAy.monitor.Position;
	FBURTKAxisMovePos(&URTKAxisMovePosY);
	if(URTKAxisMovePosY.enable)
	URTKAy.control.U = URTKAxisMovePosY.U;

	URTKAxisMovePosZ.homing_done=URTKAxisHomeZ.done;
	URTKAxisMovePosZ.act_position=URTKAz.monitor.Position;
	FBURTKAxisMovePos(&URTKAxisMovePosZ);
	if(URTKAxisMovePosZ.enable)
	URTKAz.control.U = URTKAxisMovePosZ.U;

	FBURTKAxis(&URTKAx);
	FBURTKAxis(&URTKAy);
	FBURTKAxis(&URTKAz);
	*/
	URTK_Ctrl.Ustator=0;
	//FBURTKCtrl(&URTK_Ctrl);
	if(BtnS){
		URTK_Ctrl.Ustator=32767;
		//URTK_Ctrl.AxisZ.hardware.PulseWidthCurrentPWM = 24575;
	}
	//
	if (!homing)
	{
		URTK_Ctrl.AxisY.hardware.PulseWidthCurrentPWM = 32000;
		if (URTK_Ctrl.AxisY.hardware.StatusInputP)
		{
			homing = 1;
			URTK_Ctrl.FBHomingY.ResetCounter = 1;
		}
	}
	else

	{
		URTK_Ctrl.FBHomingY.ResetCounter = 0;
		pos_new = URTK_Ctrl.AxisY.hardware.Counter/24*3;
		speed = (pos_new - pos_last)/0.01;

		pd.in = pos_ust - pos_new;
		FB_PD(&pd);

		pid.in = pd.out - speed;
		FB_Controller(&pid);

		integ = (INT)pid.out;

		URTK_Ctrl.AxisY.hardware.PulseWidthCurrentPWM = -integ;

		//URTK_Ctrl.Control.ManualCtrl = 1;

		if (URTK_Ctrl.AxisY.hardware.StatusInputN)
		{
			URTK_Ctrl.AxisY.hardware.PulseWidthCurrentPWM = 0;
			URTK_Ctrl.AxisY.hardware.StatusInputP = 0;
			flag = 0;
		}

		//FBURTKCtrl(&URTK_Ctrl);
		pos_last=pos_new;
	}

}

void _EXIT ProgramExit(void)
{
	// Insert code here
}
```

#### Types.typ - Local data types
```iecst
TYPE
	TState_led :
		(
		ST_Led1,
		ST_Led2,
		ST_Led3,
		ST_Led4
		);
END_TYPE
```

#### Variables.var - Local variables
```iecst
VAR
	speed : REAL;
	pos_new : REAL;
	pos_last : REAL;
	led4 : BOOL;
	led3 : BOOL;
	led2 : BOOL;
	led1 : BOOL;
	URTK_Ctrl : FBURTKCtrl;
	BtnS : BOOL;
	PageNum : INT;
	State_led : TState_led;
	cnt : INT;
	flag : BOOL := FALSE;
	I_ust : REAL;
	pid : FB_Controller;
	homing : BOOL;
	pos_ust : REAL;
	pd : FB_PD;
	integ : INT;
END_VAR
```

### Program Logical/Home (ANSIC)

#### Main.c - Initialization code
```c
#include <bur/plctypes.h>

#ifdef _DEFAULT_INCLUDES
	#include <AsDefault.h>
#endif

void _INIT ProgramInit(void)
{
	FB_URTKAxisHome(&ST_IDLE);
}

void _CYCLIC ProgramCyclic(void)
{

	if(BntC)
	{
		U_fast=24.0;

	}

}

void _EXIT ProgramExit(void)
{
	// Insert code here

}
```

#### Variables.var - Local variables
```iecst
VAR
	U_fast : REAL;
	BntC : BOOL;
	enable : BOOL;
END_VAR
```

Listed in the project but not available here: Logical/Global.typ, Logical/Global.var, Logical/Libraries/Library/FB_Motor.c, Logical/Libraries/Library/FB_Integrator.c, Logical/Libraries/Library/FB_Axis.c, Logical/Libraries/URTK_lib/Constants.var, Logical/Home/Types.typ
